TYPE (* typedef of the network event structure *)
  (* Version 1.0, 2025-10-18, franz *)
  PACKAGE isobus::pgn;
  ISONETEVENT_T : STRUCT
    eNetEvent : USINT := ISO_NETEVENT_e::Isonet_Last; (* Which event occurs in the network member administration? *)
    eMemberRefer : SINT := ISOUSERHOME_e::notdef; (* Which member concerned: Owner of this callback, another internal or external CF *)
    s16OwnCfHnd : INT; (* CF handle of the entry for which the callback is triggered *)
    s16Handle : INT; (* Network member handle of the CF / user (event source CF handle) *)
    u8SAMember : USINT; (* Current source address (SA) of the network member *)
    cfName : isobus::pgn::CF_NAME_T; (* ISOBUS name of the control function *)
  END_STRUCT;
END_TYPE
